FUNCTION_BLOCK E_PERMIT_1 (* permissive propagation of an event (generic FB) *)
  (* Standard: 61499-1 Annex A; Description: Copyright (c) 2017, 2026 fortiss GmbH, HR Agrartechnik GmbH This program and the accompanying materials are made available under the terms of the Eclipse Public License 2.0 which is available at https://www.eclipse.org/legal/epl-2.0/ SPDX-License-Identifier: EPL-2.0 Some portions generated by Gemini CLI *)
  (* Version 1.0, 2026-02-01, Franz Höpfinger, HR Agrartechnik GmbH, Initial creation based on E_PERMIT and E_SPLIT_3 *)
  PACKAGE iec61499::events;
  {SET_ATTRIBUTE(eclipse4diac::core::GenericClassName, 'GEN_E_PERMIT')}
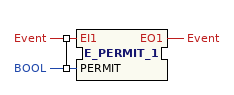
  EVENT_INPUT
    EI1 WITH PERMIT; (* Event input 1 *)
  END_EVENT
  EVENT_OUTPUT
    EO1; (* Event output 1 *)
  END_EVENT
  VAR_INPUT
    PERMIT : BOOL; (* Permit event *)
  END_VAR
END_FUNCTION_BLOCK
